# EPICS StreamDevice protocol: spsioc/Aml_Gauge.proto
# amlGauge.proto
# Proto file for the AML NGC2D Gauge Controller
# Mehmet Bozdogan 10/11/2017
#
################################################################################
OutTerminator = CR LF;
InTerminator  = CR LF;
ReadTimeout = 1000;
WriteTimeout = 1000;
PollPeriod = 1000;
ReplyTimeout = 1000;
LockTimeout = 5000;
ExtraInput = Ignore;

getStatus
{
	out "*S0";
	wait 200;
	in	"%*9r"
		"%*7r"
		","
		"%*41r";
}

getPresIG
{
	out "*S0";
	wait 200;
	in "%*9r"
	   "%e"
	   ","
	   "%*41c"
	   ;
	@mismatch{
		out "*S0";
		wait 500;
		in "%*9r"
		"%e"
		","
		"%*41c"
		;
	}
}

setCtrlMode
{
	out "%{*R0|*C0}";
}
